// TIA Portal V20 export
DATA_BLOCK "PARA"   // DB16
{ S7_Optimized_Access := 'FALSE' }
VERSION : 0.1
// stored: AutoNumber true, DBAccessibleFromOPCUA true, DBAccessibleFromWebserver true, IsOnlyStoredInLoadMemory false, IsWriteProtectedInAS false
   VAR
      Machine : Struct   // [p001 - p099] 장비 파라미터
         ID : USInt := 2;   // [p1] Machine ID
         MachinType : USInt := 2;   // [p2] Machin Type
         ToolType : USInt := 2;   // [p3] Gripper Type
         LayoutType : USInt;   // [p4]
         p5 : USInt;   // [p5]
         p6 : USInt;   // [p6]
         p7 : USInt;   // [p7]
         ModuleCount : USInt := 3;   // [p8] Modele Count
         AxisCount : USInt := 4;   // [p9] AxisCount
         XLength : UInt := 3000;   // [p10] X-Axis Axis Length
         XLengthFront : UInt := 1903;   // [p11] X-Axis Axis Length Front
         XLengthRear : UInt := 1903;   // [p12] X-Axis Axis Length Rear
         AntiColMargin_Default : UInt := 100;   // [p13] Collision Margin
         AntiColMargin_XAC : UInt := 200;   // [p14] Collision Margin
         AntiColMargin_Pos : UInt := 300;   // [p15] Collision Margin
         AntiColMargin_Avoid : UInt := 400;   // [p16] Collision Margin
         p17 : UInt;   // [p17]
         p18 : UInt;   // [p18]
         p19 : UInt;   // [p19]
         Z_Drum_Turn : USInt;   // [p20] Z-Axis Drum Turn
         Z_BeltInitCount : USInt;   // [p21] Z_BeltInitCount
         Z_BeltThickness : Real;   // [p22] Z_BeltThickness
         Z_Drum_Dia : Real;   // [p23] Z-Axis Drum Diameter
         Z_GripTipHeight : Real := 10.0;   // [p24] Z-Axis GripTip Height
         p25 : Real;   // [p25]
         p26 : Real;   // [p26]
         p27 : Real;   // [p27]
         p28 : Real;   // [p28]
         p29 : Real;   // [p29]
         G_LinkBase : Real := 62.0;   // [p30] G-Axis LinkBase Length
         G_TipBase : Real := 25.6;   // [p31] G-Axis TipBase Length
         G_Link : Real := 265.0;   // [p32] G-Axis Link Length
         G_GHP : Real := 261.65;   // [p33] G-Axis GHP Length
         G_Offset : Real := 4.76;   // [p34] G-Axis ACS Offset
         G_Tip : Real := 17.0;   // [p35] G-Axis Tip Length
         G_LeadScrewPitch : Real := 20.0;   // [p36] G-Axis Lead Screw Pitch
         p37 : Real;   // [p37]
         p38 : Real;   // [p38]
         p39 : Real;   // [p39]
         p40 : Real := 60.0;   // [p40]
         p41 : Real;   // [p41]
         p42 : Real;   // [p42]
         p43 : Real;   // [p43]
         p44 : Real;   // [p44]
         p45 : Real;   // [p45]
         p46 : Real;   // [p46]
         p47 : Real;   // [p47]
         p48 : Real;   // [p48]
         p49 : Real;   // [p49]
         MotorRefTorque : Array["X".."G"] of Real;   // [p50-p53]
         p54 : Real;   // [p54]
         p55 : Real;   // [p55]
         p56 : Real;   // [p56]
         p57 : Real;   // [p57]
         p58 : Real;   // [p58]
         p59 : Real;   // [p59]
         p60 : Real;   // [p60]
         p61 : Real;   // [p61]
         p62 : Real;   // [p62]
         p63 : Real;   // [p63]
         p64 : Real;   // [p64]
         p65 : Real;   // [p65]
         p66 : Real;   // [p66]
         p67 : Real;   // [p67]
         p68 : Real;   // [p68]
         p69 : Real;   // [p69]
         p70 : Real;   // [p70]
         p71 : Real;   // [p71]
         p72 : Real;   // [p72]
         p73 : Real;   // [p73]
         p74 : Real;   // [p74]
         p75 : Real;   // [p75]
         p76 : Real;   // [p76]
         p77 : Real;   // [p77]
         p78 : Real;   // [p78]
         p79 : Real;   // [p79]
         HomeDogLen : Array["X".."G"] of Real;   // [p80-p83] Home Dog Length
         p84 : Real;   // [p84]
         p85 : Real;   // [p85]
         p86 : Real;   // [p86]
         p87 : Real;   // [p87]
         p88 : Real;   // [p88]
         p89 : Real;   // [p89]
         p90 : Real;   // [p90]
         p91 : Real;   // [p91]
         p92 : Real;   // [p92]
         p93 : Real;   // [p93]
         p94 : Real;   // [p94]
         p95 : Real;   // [p95]
         CellOriginDogLen : Array["X".."Y"] of Real;   // [p96-p97] Cell Origin Dog Len
         StandAloneRangeXMin : Real := 4300.0;   // [p98] StandAlone Range Min
         StandAloneRangeXMax : Real := 12500.0;   // [p99] StandAlone Range Max
      END_STRUCT;
      Network : Struct   // [p100 - p149] 네트워크 파라미터
         Device : Array[0..3] of Byte;
         GR1 : Array[0..3] of Byte;
         GR2 : Array[0..3] of Byte;
         GR3 : Array[0..3] of Byte;
         GCS : Array[0..3] of Byte;
         GRM : Array[0..3] of Byte;
      END_STRUCT;
      DI_Config : "GR_DI_Config";   // [p150 - p299] DI Config (Reserved 영역 포함)
      DQ_Config { S7_SetPoint := 'True'} : "GR_DQ_Config";   // [p300 - p399] DQ Config (Reserved 영역 포함)
      Sensor : Struct   // [p400 - p499] Sensor 파라미터
         ItemDetectDistance_LL : Real := 15.0;   // [p400]
         ItemDetectDistance_L : Real;   // [p401]
         ItemDetectDistance_M : Real := 300.0;   // [p402]
         ItemDetectDistance_H : Real := 800.0;   // [p403]
         LaserDiag_SpreadLimit : Real := 8.0;   // [p404] 그리퍼 레이저 진단 : 한 측정의 방향별 비드 높이 편차 폭(최대-최소) 기준 (mm). 0 이면 8
         LaserDiag_PlanarLimit : Real := 4.0;   // [p405] 그리퍼 레이저 진단 : TBR 비평면 성분 |(L+R)-(F+B)| 기준 (mm). 0 이면 4
         LaserDiag_JumpDist : Real := 20.0;   // [p406] 그리퍼 레이저 진단 : 연속 샘플 거리 급변 기준 (mm). 0 이면 20
         LaserDiag_JumpCountLimit : Real := 5.0;   // [p407] 그리퍼 레이저 진단 : 한 측정의 급변 횟수 기준 (회). 0 이면 5
         LaserDiag_ConsecLimit : Real := 3.0;   // [p408] 그리퍼 레이저 진단 : 무응답 / 불안정 연속 측정 수 알람 기준 (회). 0 이면 3
         FLD_AntiColDistance : Real := 40.0;   // [p409] FLD_AntiColDistance
         FLD_Offset : Real := 62.0;   // [p410] FLDOffset
         XACF_Offset : Real := 755.0;   // [p411] XAC_Front_Offset
         XACR_Offset : Real := 755.0;   // [p412] XAC_Rear_Offset
         GIDL_Offset : Real := 41.0;   // [p413] GDL Offset
         GIDF_Offset : Real := 41.0;   // [p414] GDF Offset
         GIDR_Offset : Real := 41.0;   // [p415] GDR Offset
         GIDB_Offset : Real := 41.0;   // [p416] GDB Offset
         GIDType : USInt;
         GIDL_ZOffset : Real;   // [p418] GDL 높이 오프셋 (mm) : 빔 높이 - 그리퍼 Z 기준. 자동 교정(LASERDIAG.ZCal) 이 기록
         GIDF_ZOffset : Real;   // [p419] GDF 높이 오프셋 (mm) : 빔 높이 - 그리퍼 Z 기준. 자동 교정(LASERDIAG.ZCal) 이 기록
         GIDR_ZOffset : Real;   // [p420] GDR 높이 오프셋 (mm) : 빔 높이 - 그리퍼 Z 기준. 자동 교정(LASERDIAG.ZCal) 이 기록
         GIDB_ZOffset : Real;   // [p421] GDB 높이 오프셋 (mm) : 빔 높이 - 그리퍼 Z 기준. 자동 교정(LASERDIAG.ZCal) 이 기록 (TBR)
         LaserDiag_BiasLimit : Real := 5.0;   // [p422] 그리퍼 레이저 진단 : 센서별 높이 편차 이동평균 알람 기준 (mm). 0 이면 5
         LaserDiag_BiasMinSamples : Real := 20.0;   // [p423] 그리퍼 레이저 진단 : 높이 편차 알람 판정 최소 측정 수 (회). 0 이면 20
         LaserDiag_BiasAlpha : Real := 0.1;   // [p424] 그리퍼 레이저 진단 : 높이 편차 이동평균 계수 (0~1). 0 이면 0.1
         LaserZCal_SampleCount : Real := 5.0;   // [p425] 레이저 Z 오프셋 자동 교정 : 측정 횟수 (회). 0 이면 5
         LaserZCal_MaxStdDev : Real := 2.0;   // [p426] 레이저 Z 오프셋 자동 교정 : 방향별 편차 표준편차 허용 (mm). 0 이면 2
         LaserZCal_MaxCorrection : Real := 20.0;   // [p427] 레이저 Z 오프셋 자동 교정 : 방향별 보정량 허용 (mm). 0 이면 20
         LaserInnerDia_Offset : Real;   // [p428] 레이저 원 맞춤 내경 보정 (mm, 부호 포함) : 측정 내경에 더함. PICK / 들어갈 때 / 나갈 때 / 수동 측정 공통, 0 = 보정 없음
         LaserFit_TbrTolerance : Real;   // [p429] TBR 4점 원 맞춤 검증 허용 (mm) : 3점 원 중심에서 4번째 점까지 거리와 반지름 차이 한계, 넘으면 FitError 3. 0 이면 3
         p430 : Real;
         X1RD_Offset : Real;   // [p431] X1RD Offset
         X2RD_Offset : Real;   // [p432] X2RD Offset
         p433 : Real;
         p434 : Real;
         p435 : Real;
         p436 : Real;
         p437 : Real;
         p438 : Real;
         p439 : Real;
         p440 : Real;
         p441 : Real;
         p442 : Real;
         p443 : Real;
         p444 : Real;
         p445 : Real;
         p446 : Real;
         p447 : Real;
         p448 : Real;
         p449 : Real;
         p450 : Real;
         p451 : Real;
         p452 : Real;
         p453 : Real;
         p454 : Real;
         p455 : Real;
         p456 : Real;
         p457 : Real;
         p458 : Real;
         p459 : Real;
         p460 : Real;
         p461 : Real;
         p462 : Real;
         p463 : Real;
         p464 : Real;
         p465 : Real;
         p466 : Real;
         p467 : Real;
         p468 : Real;
         p469 : Real;
         p470 : Real;
         p471 : Real;
         p472 : Real;
         p473 : Real;
         p474 : Real;
         p475 : Real;
         p476 : Real;
         p477 : Real;
         p478 : Real;
         p479 : Real;
         p480 : Real;
         p481 : Real;
         p482 : Real;
         p483 : Real;
         p484 : Real;
         p485 : Real;
         p486 : Real;
         p487 : Real;
         p488 : Real;
         p489 : Real;
         p490 : Real;
         p491 : Real;
         p492 : Real;
         p493 : Real;
         p494 : Real;
         p495 : Real;
         p496 : Real;
         p497 : Real;
         p498 : Real;
         p499 : Real;
      END_STRUCT;
      Drive : Struct   // [p500 - p899] Drive
         SpeedFactor : Array["X".."G"] of Real;   // [p500-p515] 축 속도 배율 %
         PIN : Array["X".."G"] of Real;   // [p516-p531] 축 정위치 범위
         PIH : Array["X".."G"] of Real;   // [p532-p547] 축 정위치 해제 범위
         StandStillSpd : Array["X".."G"] of Real;   // [p548-p563]축 정지 결정 속도 (m/s) 파라미터
         StandStillDwellTime : Array["X".."G"] of Real;   // [p564-p579] 축 정지 결정 시간 파라미터
         FaultMargin : Array["X".."G"] of Real;   // [p580-p595] 축 포지셔닝 명령 허용 오차 파라미터(mm)
         JogTorqLimit : Array["X".."G"] of Real;   // [p596-p611] 축 조그 기동 시 토크 리미트(%) 파라미터
         InverseHomingDir : Array["X".."G"] of USInt;   // [p612-p627] Homing 방향 변경 파라메터
         RangeMin : Array["X".."G"] of Real;   // [p628-p643] 축 가동 최소 범위
         RangeMax : Array["X".."G"] of Real;   // [p644-p659] 축 가동 최소 범위
         HomePos : Array["X".."G"] of Real;   // [p660-p675] 축 홈 위치
         MaintPos : Array["X".."G"] of Real;   // [p676-p691] 축 Maintenance 위치
         UtilityPos_A : Array["X".."G"] of Real;   // [p692-p707] Utility Pos A
         UtilityPos_B : Array["X".."G"] of Real;   // [p708-p723] Utility Pos B
         CellOriginPos : Array["X".."Y"] of Real;   // [p756-p757] Cell Layout 원점
         SyncFltDiff : Real := 30.0;   // [p772] X1, X2축 동기 오차 Fault 거리 파라미터
         SyncFltDiffMarginByVelocity : Real := 40.0;   // [p773] X1, X2축 동기 오차 Fault 감지 거리 속도 마진 파라미터
         OriginPos : Array["X".."G"] of Real;   // [p784..p799] 드라이브 원점 위치 (ACS)
         MCS_TO_ACS : Array["X".."G", 0..2] of Real;   // [p800..p849] ACS 변환 계수
         ACS_TO_MCS : Array["X".."G", 0..2] of Real;   // [p850..p899] MCS 변환 계수
      END_STRUCT;
      Task : Struct   // [p900 - p999] Task
         CheckStation : Bool := TRUE;   // [p900] 명령 수행 시 Station Interlock 확인 여부 파라미터
         CheckGoods : Bool := TRUE;   // [p901] 명령 수행 시 물체 감지 센서 사용 여부, PICK 인 경우 타이어 빠짐 Detection
         CheckCellUse : Bool := TRUE;   // [p902] 명령 수행 시 Cell 사용 여부 파라미터
         CheckCollision : Bool := TRUE;   // [p903] 명령 수행 시 충돌방지 로직 사용 여부 파라미터
         EnablePreGrip : Bool := TRUE;   // [p904] 명령 수행 시 PreGrip 사용 여부, PreGrip : PICK 명령 시 Gripper 를 PreGripDelta 거리 만큼 미리 이동 시키는 기능
         EnableCreepUp : Bool := TRUE;   // [p905] PICK 명령 수행 이후 저속 들기 사용 여부 파라미터
         EnableCreepDown : Bool := TRUE;   // [p906] DROP 명령 수행 시 저속 내려 놓기 사용 여부 파라미터
         EnableTorqBack : Bool := TRUE;   // [p907] 명령 수행 시 일정 구간 Gripper TorqRelease 사용 여부 파라미터
         EnableInitializingBeforeAuto : Bool;   // [p908] 명령 수행 전 Initializing 확인 여부 파라미터
         p909 : Bool;   // [p909]
         p910 : Bool;   // [p910]
         p911 : Bool;   // [p911]
         p912 : Bool;   // [p912]
         p913 : Bool;   // [p913]
         p914 : Bool;   // [p914]
         p915 : Bool;   // [p915]
         p916 : Bool;   // [p916]
         p917 : Bool;   // [p917]
         p918 : Bool;   // [p918]
         p919 : Bool;   // [p919]
         p920 : Bool;   // [p920]
         p921 : Bool;   // [p921]
         p922 : Bool;   // [p922]
         p923 : Bool;   // [p923]
         p924 : Bool;   // [p924]
         p925 : Bool;   // [p925]
         p926 : Bool;   // [p926]
         p927 : Bool;   // [p927]
         p928 : Bool;   // [p928]
         p929 : Bool;   // [p929]
         BlendingDistance : Real := 500.0;   // [p930] XYZ 블랜딩 거리(mm) 파라미터
         MoveAllowZHeight : Real := 2700.0;   // [p931] XY 동작 허용 Z 높이(mm) 파라미터
         StationGoodsGap : Real := 20.0;   // [p932] Station 다스택 적재 시 타이어 간의 거리 파라미터
         StationDragDistance : Real := 100.0;   // [p933] Station 명령 시 Drag 이동 거리 파라미터
         StationDragHeight : Real := 500.0;   // [p934] Station 명령 시 Drag 동작 시작 높이 파라미터
         StationDragBlendDistance : Real := 200.0;   // [p935] Station 명령시 Drage 동작 Blending 거리 파라미터
         PickSlowDownDistance : Real := 150.0;   // [p936] PICK 명령 수행 저속 운행 거리 여부 파라미터
         DropSlowDownDistance : Real := 150.0;   // [p937] DROP 명령 수행 저속 운행 거리 여부 파라미터
         DropOffset : Real := 10.0;   // [p938] DROP 명령 수행 시 Z축 DROP 포지션 Offset 파라미터, 지정된 포지션 + Offset 위치에 DROP 명령을 수행 하게 됨
         PreGripDelta : Real := 100.0;   // [p939] 명령 수행 중 PREGRIP시 타이어와의 거리 파라미터
         G_DropTorq_Factor : Real := 70.0;   // [p940] DROP 명령 수행 시 Gripper Torq(%) 파라미터
         G_PickTorq_Factor : Real := 50.0;   // [p941] PICK 명령 수행 시 Gripper Torq(%) 파라미터
         G_TorqLimitAllowDistance : Real := 10.0;   // [p942] Gripper Torq 리미트 동작 시 Inposition 허용 거리(mm) 파라미터
         G_TorqRelease_Factor : Real := 100.0;   // [p943] Gripper Torq Release 동작시 토크 제한 해제 % 파라미터
         G_TorqReleaseRemainZHeight : Real := 50.0;   // [p944] Gripper Torq Release 동작 높이 (mm) 파라미터
         G_PickGripOffset : Real;   // [p945] Gripper PICK 명령시 Gripper Position Offset (mm) 파라미터
         G_PickGripOffset_Factor : Real;   // [p946] Gripper PICK 명령시 Gripper Position Offset (%) 파라미터, 명령 Position에 대한 추가 %를 의미한다
         PreDropHeight_Factor : Real;   // [p947] PreGrip Drop시 명령시 시작 Z 위치
         PrePickHeight_Factor : Real;   // [p948] PreGrip Pick 명령시 타이어 높이 대비 시작 위치 %
         G_TorqDetect_OnRatio : Real := 90.0;   // [p949] Gripper 토크 검출 켜짐 기준(%) 파라미터, 적용 중 토크 제한값 대비. 0 이면 90
         G_TorqDetect_OffRatio : Real := 70.0;   // [p950] Gripper 토크 검출 꺼짐 기준(%) 파라미터, 적용 중 토크 제한값 대비. 0 이면 70
         G_TorqDetect_DwellTime : Real := 0.2;   // [p951] Gripper 토크 검출 켜짐 유지시간(s) 파라미터. 0 이면 0.2
         G_MeasureTorq_Factor : Real;   // [p952] 토크 내경 측정 시 Gripper 토크 제한(%) 파라미터. 0 이면 기존값 (자동 측정 G_PickTorq_Factor, 수동 측정 15)
         G_MeasureTorq_Offset : Real;   // [p953] 토크 내경 측정(자동, MeasureItem) 보정 (mm, 부호 포함) : 반복 평균 G 위치에 더함. 0 = 보정 없음 (기존 고정값 -5)
         G_MeasureTorq_OffsetManual : Real;   // [p954] 토크 내경 측정(수동) 보정 (mm, 부호 포함) : 토크 도달 G 위치에 더함. 0 = 보정 없음 (기존 고정값 -8)
         p955 : Real;   // [p955]
         p956 : Real;   // [p956]
         p957 : Real;   // [p957]
         p958 : Real;   // [p958]
         p959 : Real;   // [p959]
         pickRetryCountMax : USInt := 1;   // [p960]
         p961 : Real;   // [p961]
         p962 : Real;   // [p962]
         p963 : Real;   // [p963]
         p964 : Real;   // [p964]
         p965 : Real;   // [p965]
         p966 : Real;   // [p966]
         p967 : Real;   // [p967]
         p968 : Real;   // [p968]
         p969 : Real;   // [p969]
         Pick_GripExtra : Real;   // [p970]
         Pick_GripBackDelta : Real;   // [p971]
         GripBackMin : Real;   // [p972] Pick Drop 시 폈다 오므리는 동작시 오므릴때 내경값 -n 제한
         p973 : Real;   // [p973]
         p974 : Real;   // [p974]
         p975 : Real;   // [p975]
         p976 : Real;   // [p976]
         p977 : Real;   // [p977]
         p978 : Real;   // [p978]
         p979 : Real;   // [p979]
         p980 : Real;   // [p980]
         p981 : Real;   // [p981]
         p982 : Real;   // [p982]
         p983 : Real;   // [p983]
         p984 : Real;   // [p984]
         p985 : Real;   // [p985]
         p986 : Real;   // [p986]
         p987 : Real;   // [p987]
         p988 : Real;   // [p988]
         p989 : Real;   // [p989]
         p990 : Real;   // [p990]
         p991 : Real;   // [p991]
         p992 : Real;   // [p992]
         p993 : Real;   // [p993]
         p994 : Real;   // [p994]
         p995 : Real;   // [p995]
         p996 : Real;   // [p996]
         p997 : Real;   // [p997]
         p998 : Real;   // [p998]
         p999 : Real;   // [p999]
      END_STRUCT;
      Timeout : Struct   // [p1000 - p1099] Timout
         PowerOn : Real := 1.0;   // [p1000] PowerOn 단계에서 TimeOut (ms) 파라미터, 1000ms = 1.0s
         DriveOn : Real := 3.0;   // [p1001] DriveOn 단계에서 TimeOut (ms) 파라미터, 1000ms = 1.0s
         DriveOffDly : Real := 60.0;   // [p1002] IDLE 상태에서 Drive Off 동작 타이머(ms), 1000ms = 1.0s
         DriveOffDlyForJog : Real := 5.0;   // [p1003] Manual, JOG 동작 시 Drive Off 동작 타이머(ms), 1000ms = 1.0s
         DriveReady : Real := 0.5;   // [p1004] 명령 실행 전 DriveReady TimeOut 파라미터(ms), 1000ms=1.0s
         p1005 : Real;
         p1006 : Real;
         p1007 : Real;
         p1008 : Real;
         p1009 : Real;
         SetOrigin : Array["X".."X2"] of Real;   // [p1010-p1025] 축 원점 이동 Timeout
         p1026 : Real;   // [p1026]
         p1027 : Real;   // [p1027]
         p1028 : Real;   // [p1028]
         p1029 : Real;   // [p1029]
         BeltTentionOnDlyTime : Real := 0.3;   // [p1030]
         p1031 : Real;   // [p1031]
         p1032 : Real;   // [p1032]
         p1033 : Real;   // [p1033]
         p1034 : Real;   // [p1034]
         p1035 : Real;   // [p1035]
         p1036 : Real;   // [p1036]
         p1037 : Real;   // [p1037]
         p1038 : Real;   // [p1038]
         p1039 : Real;   // [p1039]
         p1040 : Real;   // [p1040]
         p1041 : Real;   // [p1041]
         p1042 : Real;   // [p1042]
         p1043 : Real;   // [p1043]
         p1044 : Real;   // [p1044]
         p1045 : Real;   // [p1045]
         p1046 : Real;   // [p1046]
         p1047 : Real;   // [p1047]
         p1048 : Real;   // [p1048]
         p1049 : Real;   // [p1049]
         p1050 : Real;   // [p1050]
         p1051 : Real;   // [p1051]
         p1052 : Real;   // [p1052]
         p1053 : Real;   // [p1053]
         p1054 : Real;   // [p1054]
         p1055 : Real;   // [p1055]
         p1056 : Real;   // [p1056]
         p1057 : Real;   // [p1057]
         p1058 : Real;   // [p1058]
         p1059 : Real;   // [p1059]
         CVInterlock : Real := 30.0;   // [p1060] Station InterLock TimOut 파라미터(ms), 1000ms=1.0s
         p1061 : Real;   // [p1061]
         p1062 : Real;   // [p1062]
         p1063 : Real;   // [p1063]
         p1064 : Real;   // [p1064]
         p1065 : Real;   // [p1065]
         p1066 : Real;   // [p1066]
         p1067 : Real;   // [p1067]
         p1068 : Real;   // [p1068]
         p1069 : Real;   // [p1069]
         p1070 : Real;   // [p1070]
         p1071 : Real;   // [p1071]
         p1072 : Real;   // [p1072]
         p1073 : Real;   // [p1073]
         p1074 : Real;   // [p1074]
         p1075 : Real;   // [p1075]
         p1076 : Real;   // [p1076]
         p1077 : Real;   // [p1077]
         p1078 : Real;   // [p1078]
         p1079 : Real;   // [p1079]
         p1080 : Real;   // [p1080]
         p1081 : Real;   // [p1081]
         p1082 : Real;   // [p1082]
         p1083 : Real;   // [p1083]
         p1084 : Real;   // [p1084]
         p1085 : Real;   // [p1085]
         p1086 : Real;   // [p1086]
         p1087 : Real;   // [p1087]
         p1088 : Real;   // [p1088]
         p1089 : Real;   // [p1089]
         CommGRM : Real := 3.0;   // [p1090] Mainpanel 통신 TimeOut 파라미터(ms),1000ms=1.0s
         CommGCS : Real;   // [p1091] GCS 통신 TimeOut 파라미터(ms),1000ms=1.0s
         CommFrontGR : Real;   // [p1092] GCS 통신 TimeOut 파라미터(ms),1000ms=1.0s
         CommRearGR : Real;   // [p1093] GCS 통신 TimeOut 파라미터(ms),1000ms=1.0s
         p1094 : Real;   // [p1094]
         p1095 : Real;   // [p1095]
         p1096 : Real;   // [p1096]
         p1097 : Real;   // [p1097]
         CsvImport : Real := 10.0;   // [p1098] 파라미터 파일(CSV) 읽기 TimeOut 파라미터(s)
         CsvExport : Real := 10.0;   // [p1099] 파라미터 파일(CSV) 쓰기 TimeOut 파라미터(s)
      END_STRUCT;
      SpeedSet : Array["X".."G", 0..9] of "LGR_PARA_SpeedSet";   // [p1100 - p1799] SpeedSet
   END_VAR
BEGIN
   Machine.MotorRefTorque[1] := 69.0;
   Machine.MotorRefTorque[2] := 45.0;
   Machine.MotorRefTorque[3] := 68.0;
   Machine.MotorRefTorque[4] := 6.5;
   Machine.HomeDogLen[1..2] := 20.0;
   Machine.HomeDogLen[3] := 40.0;
   Machine.HomeDogLen[4] := 4.0;
   Machine.CellOriginDogLen[1..2] := 20.0;
   Network.Device[0] := 16#00C0;
   Network.Device[1] := 16#00A8;
   Network.Device[2] := 16#0001;
   Network.Device[3] := 16#0066;
   Network.GR1[0] := 16#00C0;
   Network.GR1[1] := 16#00A8;
   Network.GR1[2] := 16#0001;
   Network.GR1[3] := 16#0065;
   Network.GR2[0] := 16#00C0;
   Network.GR2[1] := 16#00A8;
   Network.GR2[2] := 16#0001;
   Network.GR2[3] := 16#0066;
   Network.GR3[0] := 16#00C0;
   Network.GR3[1] := 16#00A8;
   Network.GR3[2] := 16#0001;
   Network.GR3[3] := 16#0067;
   Network.GCS[0] := 16#00C0;
   Network.GCS[1] := 16#00A8;
   Network.GCS[2] := 16#000A;
   Network.GCS[3] := 16#0096;
   Network.GRM[0] := 16#00C0;
   Network.GRM[1] := 16#00A8;
   Network.GRM[2] := 16#0001;
   Network.GRM[3] := 16#0064;
   Drive.SpeedFactor[1..4] := 1.0;
   Drive.PIN[1] := 3.0;
   Drive.PIN[2..3] := 1.0;
   Drive.PIN[4] := 0.2;
   Drive.PIH[1..2] := 2.0;
   Drive.PIH[3..4] := 1.0;
   Drive.StandStillSpd[1..3] := 0.5;
   Drive.StandStillSpd[4] := 4.0;
   Drive.StandStillDwellTime[1..4] := 0.1;
   Drive.FaultMargin[1] := 2.0;
   Drive.FaultMargin[2..4] := 0.2;
   Drive.JogTorqLimit[1..2] := 50.0;
   Drive.JogTorqLimit[3..4] := 100.0;
   Drive.RangeMin[1] := 4300.0;
   Drive.RangeMin[2] := 928.0;
   Drive.RangeMin[3] := 60.0;
   Drive.RangeMin[4] := 295.0;
   Drive.RangeMax[1] := 12500.0;
   Drive.RangeMax[2] := 9428.0;
   Drive.RangeMax[3] := 3279.9;
   Drive.RangeMax[4] := 630.0;
   Drive.HomePos[1] := 15000.0;
   Drive.HomePos[2] := 1000.0;
   Drive.HomePos[3] := 3279.9;
   Drive.HomePos[4] := 271.41;
   Drive.MaintPos[1] := 15000.0;
   Drive.MaintPos[2] := 1000.0;
   Drive.MaintPos[3] := 600.0;
   Drive.MaintPos[4] := 630.0;
   Drive.UtilityPos_A[1] := 15000.0;
   Drive.UtilityPos_A[2] := 1000.0;
   Drive.UtilityPos_A[4] := 275.0;
   Drive.UtilityPos_B[4] := 630.0;
   Drive.CellOriginPos[1] := 5700.0;
   Drive.CellOriginPos[2] := 1639.6;
   Drive.OriginPos[1..2] := 1000.0;
   Drive.OriginPos[3] := 3300.0;
   Drive.OriginPos[4] := 271.41;
   Drive.MCS_TO_ACS[1,1] := 1.0;
   Drive.MCS_TO_ACS[2,1] := 1.0;
   Drive.MCS_TO_ACS[2,2] := 66.0;
   Drive.MCS_TO_ACS[3,0] := -6.15498E-06;
   Drive.MCS_TO_ACS[3,1] := 0.9892772;
   Drive.MCS_TO_ACS[3,2] := 121.0;
   Drive.MCS_TO_ACS[4,1] := 1.0;
   Drive.ACS_TO_MCS[1,1] := 1.0;
   Drive.ACS_TO_MCS[2,1] := 1.0;
   Drive.ACS_TO_MCS[2,2] := -66.0;
   Drive.ACS_TO_MCS[3,0] := 6.77245E-06;
   Drive.ACS_TO_MCS[3,1] := 1.008633;
   Drive.ACS_TO_MCS[3,2] := -122.0;
   Drive.ACS_TO_MCS[4,1] := 1.0;
   Timeout.SetOrigin[1] := 1.0;
   Timeout.SetOrigin[2] := 2.0;
   Timeout.SetOrigin[3] := 8.0;
   Timeout.SetOrigin[4..6] := 1.0;
   SpeedSet[1,0].Speed := 20.0;
   SpeedSet[1,1].Speed := 50.0;
   SpeedSet[1,2].Speed := 1000.0;
   SpeedSet[1,3].Speed := 2000.0;
   SpeedSet[1,4].Speed := 4000.0;
   SpeedSet[1,5].Speed := 400.0;
   SpeedSet[1,6].Speed := 20.0;
   SpeedSet[1,7].Speed := 5.0;
   SpeedSet[2,0].Speed := 20.0;
   SpeedSet[2,1].Speed := 50.0;
   SpeedSet[2,2].Speed := 1000.0;
   SpeedSet[2,3].Speed := 2000.0;
   SpeedSet[2,4].Speed := 4000.0;
   SpeedSet[2,5].Speed := 400.0;
   SpeedSet[2,6].Speed := 20.0;
   SpeedSet[2,7].Speed := 5.0;
   SpeedSet[3,0].Speed := 20.0;
   SpeedSet[3,1].Speed := 100.0;
   SpeedSet[3,2].Speed := 1000.0;
   SpeedSet[3,3].Speed := 1250.0;
   SpeedSet[3,4].Speed := 2500.0;
   SpeedSet[3,5].Speed := 500.0;
   SpeedSet[3,6].Speed := 20.0;
   SpeedSet[3,7].Speed := 10.0;
   SpeedSet[4,0].Speed := 5.0;
   SpeedSet[4,1..2].Speed := 10.0;
   SpeedSet[4,3].Speed := 100.0;
   SpeedSet[4,4..5].Speed := 200.0;
   SpeedSet[4,6].Speed := 5.0;
   SpeedSet[4,7].Speed := 10.0;
   SpeedSet[1,0..1].Accel := 100.0;
   SpeedSet[1,2..5].Accel := 2500.0;
   SpeedSet[1,6].Accel := 500.0;
   SpeedSet[1,7].Accel := 100.0;
   SpeedSet[1,8].Accel := 2500.0;
   SpeedSet[1,9].Accel := 3000.0;
   SpeedSet[2,0..1].Accel := 100.0;
   SpeedSet[2,2..5].Accel := 2500.0;
   SpeedSet[2,6..7].Accel := 500.0;
   SpeedSet[2,8].Accel := 2500.0;
   SpeedSet[2,9].Accel := 3000.0;
   SpeedSet[3,0..1].Accel := 100.0;
   SpeedSet[3,2].Accel := 2500.0;
   SpeedSet[3,3..5].Accel := 4000.0;
   SpeedSet[3,6..7].Accel := 500.0;
   SpeedSet[3,8..9].Accel := 4000.0;
   SpeedSet[4,0..1].Accel := 100.0;
   SpeedSet[4,2].Accel := 1000.0;
   SpeedSet[4,3..5].Accel := 2500.0;
   SpeedSet[4,6..7].Accel := 1000.0;
   SpeedSet[4,8].Accel := 2500.0;
   SpeedSet[4,9].Accel := 3000.0;
   SpeedSet[1,0..1].Decel := 100.0;
   SpeedSet[1,2..5].Decel := 2500.0;
   SpeedSet[1,6].Decel := 500.0;
   SpeedSet[1,7].Decel := 100.0;
   SpeedSet[1,8].Decel := 2500.0;
   SpeedSet[1,9].Decel := 3000.0;
   SpeedSet[2,0..1].Decel := 100.0;
   SpeedSet[2,2..5].Decel := 2500.0;
   SpeedSet[2,6..7].Decel := 500.0;
   SpeedSet[2,8].Decel := 2500.0;
   SpeedSet[2,9].Decel := 3000.0;
   SpeedSet[3,0..1].Decel := 100.0;
   SpeedSet[3,2].Decel := 2500.0;
   SpeedSet[3,3..5].Decel := 4000.0;
   SpeedSet[3,6..7].Decel := 500.0;
   SpeedSet[3,8..9].Decel := 4000.0;
   SpeedSet[4,0..1].Decel := 100.0;
   SpeedSet[4,2].Decel := 1000.0;
   SpeedSet[4,3..5].Decel := 2500.0;
   SpeedSet[4,6..7].Decel := 1000.0;
   SpeedSet[4,8].Decel := 2500.0;
   SpeedSet[4,9].Decel := 3000.0;
   SpeedSet[1,0..1].JerkTime := 100.0;
   SpeedSet[1,2..5].JerkTime := 1000.0;
   SpeedSet[1,6].JerkTime := 200.0;
   SpeedSet[1,7].JerkTime := 100.0;
   SpeedSet[1,8..9].JerkTime := 1000.0;
   SpeedSet[2,0..1].JerkTime := 50.0;
   SpeedSet[2,2].JerkTime := 1000.0;
   SpeedSet[2,3..4].JerkTime := 500.0;
   SpeedSet[2,5].JerkTime := 1000.0;
   SpeedSet[2,6].JerkTime := 200.0;
   SpeedSet[2,7].JerkTime := 100.0;
   SpeedSet[2,8..9].JerkTime := 500.0;
   SpeedSet[3,0].JerkTime := 50.0;
   SpeedSet[3,1..9].JerkTime := 200.0;
   SpeedSet[4,0..1].JerkTime := 50.0;
   SpeedSet[4,2].JerkTime := 100.0;
   SpeedSet[4,3].JerkTime := 200.0;
   SpeedSet[4,4].JerkTime := 100.0;
   SpeedSet[4,5].JerkTime := 200.0;
   SpeedSet[4,6].JerkTime := 50.0;
   SpeedSet[4,7].JerkTime := 100.0;
   SpeedSet[4,8].JerkTime := 200.0;
   SpeedSet[4,9].JerkTime := 100.0;
END_DATA_BLOCK
